TYPE ST_FSM_Params :
STRUCT
	tStoppingDelay	:	TIME	:=	T#2S;
END_STRUCT
END_TYPE

(* stored: Version 1.1.0.1
   DUT ST_FSM_Params: Id {429f9595-524c-0f68-156f-621e42828ef9} *)
